{attribute 'linkalways'} 
{attribute 'no_explicit_call' := 'This FB is a CLASS and must be accessed using methods or properties'}
{attribute 'enable_dynamic_creation'}
FUNCTION_BLOCK InstanceRemovedEvent EXTENDS Event IMPLEMENTS I_InstanceRemovedEvent
VAR
	_instance : I_Instance;
END_VAR

PROPERTY PUBLIC Instance : I_Instance
GET
Instance := _instance;
END_GET
END_PROPERTY

METHOD PUBLIC Notify
VAR_INPUT
	Instance : I_Instance;
END_VAR
_instance := instance;
NotifySubscribers();
END_METHOD

END_FUNCTION_BLOCK

(* stored: Version 1.1.0.1, ProductVersion 3.1.4024.12
   POU InstanceRemovedEvent: Id {b292b512-a26a-0ae7-2b75-73ad45f338cf}, SpecialFunc None
   Property Instance: Id {8fc8a055-7f05-0f46-362c-6b87724bccf5}
   Get Get: Id {de96d4f2-6ab3-072e-25dd-23806ecf0613}
   Method Notify: Id {aff55f9e-5ab1-0257-25c1-4836cee77825} *)
